VAR_GLOBAL CONSTANT
	cRECVDATACHANNELBUFFER: INT := 20;
END_VAR

(* stored: Version 1.1.0.1, ProductVersion 3.1.0.36
   GVL IdBaseConst: Id {edf4ab20-67eb-445f-b700-5b87d1060a60} *)
